// TIA Portal V19 export
TYPE "IFM_LDL_IO"
   STRUCT
      Value_c : Real;   // Conductivity
      Value_t : Real;   // Temperature
      O_DI4 : Bool;   // Port pin 4
      O_DI2 : Bool;   // Port pin 2
      O_DA : Bool;   // Device Attached
      O_DE : Bool;   // Device Error
      O_PQ : Bool;   // Value Valid
   END_STRUCT;
END_TYPE
